// TwinCAT 3 PLC project PLC1
// ProgramVersion: 3.1.4023.0
// libraries:
//   Tc2_ControllerToolbox, * (Beckhoff Automation GmbH)
//   Tc2_Standard, * (Beckhoff Automation GmbH)
//   Tc2_System, * (Beckhoff Automation GmbH)
//   Tc3_Module, * (Beckhoff Automation GmbH)
//   VisuSymbols,3.5.10.0,System
// project tree:
//   / GlobalTextList.TcGTLO, PlcTask.TcTTO, Visualization Manager.TcVMO (not stored)
//   GVLs/ PID_DATA.TcGVL
//   POUs/ MAIN.TcPOU, PID.TcPOU, ClearPID.TcPOU
//   VISUs/ VISU1.TcVIS
// real-time tasks:
//   TASK PlcTask: cycle T#1ms, priority 20, ADS port 350
// I/O:
//   DEVICE Device 4 (EtherCAT), AmsNetId 192.168.56.1.5.1
//     Box 1 (Q.station 101 T) [Q.station 101 T]
//     Box 2 (LAN9252_STM32) [LAN9252_STM32]
// variable links:
//   PLC1/PLC1 Instance <-> Device 4 (EtherCAT)/Box 1 (Q.station 101 T)
//     PlcTask Inputs/MAIN.AIN1 <-> TxPDO mapping - Encoder/Encoder
//   PLC1/PLC1 Instance <-> Device 4 (EtherCAT)/Box 2 (LAN9252_STM32)
//     PlcTask Outputs/MAIN.Enable <-> MotorStatus/MotorStatus
//     PlcTask Outputs/MAIN.OUT <-> pwm/pwm

CONFIGURATION PLC1
    RESOURCE PLC ON TwinCAT3
        TASK PlcTask(INTERVAL := T#1ms, PRIORITY := 20);
        PROGRAM MAIN WITH PlcTask : MAIN;
    END_RESOURCE
END_CONFIGURATION

// ---- GVLs/PID_DATA.TcGVL
{attribute 'qualified_only'}
VAR_GLOBAL
	ge0 : REAL := 0;
	ge1 : REAL := 0;
	ge2 : REAL := 0;
	gu0 : REAL := 0;
	gu1 : REAL := 0;
	gp : REAL := 0.01;
	gi : REAL := 0.005;
	gd : REAL := 0;
	gset : REAL := 360;
	gmea : REAL := 0;
	gstime: REAL := 0.001;
END_VAR

// ---- POUs/MAIN.TcPOU
PROGRAM MAIN
VAR
	AIN1 AT %I*: REAL;
	OUT AT %Q*: REAL;
	Start: BOOL;
	Stop: BOOL;
	Enable: BOOL;
	
END_VAR

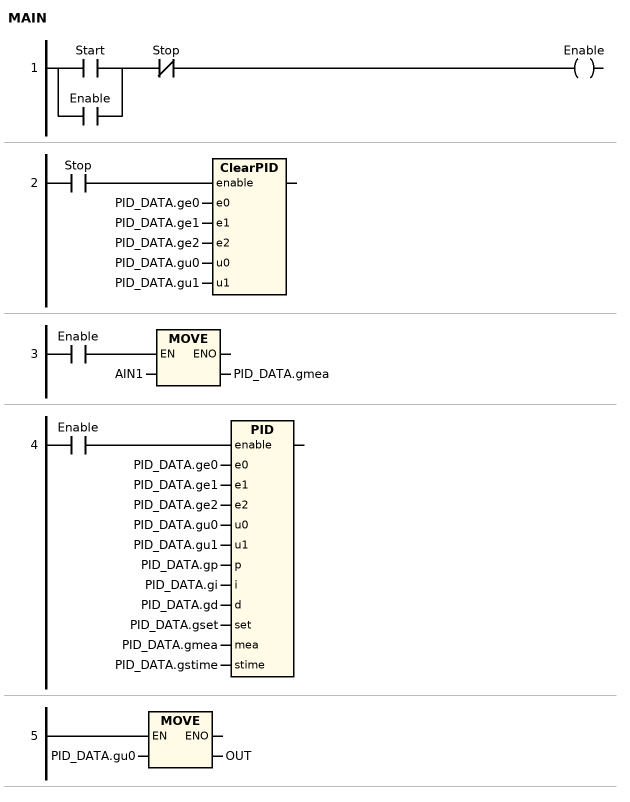
// NETWORK 1
Enable := (Start OR Enable) AND NOT Stop;

// NETWORK 2
ClearPID(enable := Stop, e0 := PID_DATA.ge0, e1 := PID_DATA.ge1, e2 := PID_DATA.ge2, u0 := PID_DATA.gu0, u1 := PID_DATA.gu1);

// NETWORK 3
IF Enable THEN PID_DATA.gmea := AIN1; END_IF

// NETWORK 4
PID(enable := Enable, e0 := PID_DATA.ge0, e1 := PID_DATA.ge1, e2 := PID_DATA.ge2, u0 := PID_DATA.gu0, u1 := PID_DATA.gu1, p := PID_DATA.gp, i := PID_DATA.gi, d := PID_DATA.gd, set := PID_DATA.gset, mea := PID_DATA.gmea, stime := PID_DATA.gstime);

// NETWORK 5
OUT := PID_DATA.gu0;

END_PROGRAM

// ---- POUs/ClearPID.TcPOU
FUNCTION ClearPID 
VAR_INPUT
	enable: BOOL;
	
END_VAR
VAR_IN_OUT
	e0, e1, e2: REAL;
	u0, u1: REAL;
	
END_VAR
VAR
END_VAR

IF (enable = TRUE) THEN
	e0 := 0;
	e1 := 0;
	e2 := 0;
	u0 := 0;
	u1 := 0;
END_IF

END_FUNCTION

// ---- POUs/PID.TcPOU
FUNCTION PID 
VAR_INPUT
	enable: BOOL;
	
END_VAR
VAR_IN_OUT
	e0, e1, e2: REAL;
	u0, u1: REAL;
	p, i, d: REAL;
	set, mea: REAL;
	stime: REAL;
	
END_VAR
VAR
END_VAR

IF (enable = TRUE) THEN
	e2 := e1;
	e1 := e0;
	e0 := set - mea;
	u1 := u0;
	u0 := u1 + p*(e0 - e1) + i*stime*(e0 + e1)/2.0 + d*(e0 - 2*e1 + e2)/stime;
END_IF

END_FUNCTION

// ---- GlobalTextList.TcGTLO
TEXTLIST GlobalTextList
  194 = '%5.4f'
  988 = 'Control'
  32 = 'Control Signal'
  512 = 'D'
  918 = 'I'
  85 = 'Measure'
  284 = 'P'
  378 = 'Setpoint'
  46 = 'Start'
  804 = 'Stop'
END_TEXTLIST

// ---- VISUs/VISU1.TcVIS
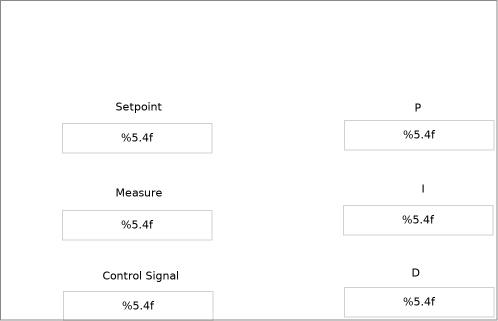
VISUALIZATION VISU1  // 498x321
    Textfield (62,210 150x30), "%5.4f", text variable: MAIN.AIN1/40.0
    Textfield (63,291 150x30), "%5.4f", text variable: MAIN.OUT
    Label (64,178 150x30), "Measure"
    Label (66,261 150x30), "Control Signal"
    Textfield (62,123 150x30), "%5.4f", text variable: PID_DATA.gset/40.0
    Label (64,92 150x30), "Setpoint"
    Textfield (343,205 150x30), "%5.4f", text variable: PID_DATA.gi
    Textfield (344,287 150x30), "%5.4f", text variable: PID_DATA.gd
    Textfield (344,120 150x30), "%5.4f", text variable: PID_DATA.gp
    Label (348,174 150x30), "I"
    Label (343,93 150x30), "P"
    Label (341,258 150x30), "D"
END_VISUALIZATION
